FUNCTION_BLOCK FB_PowerNC IMPLEMENTS I_Power
VAR_INPUT
END_VAR
VAR_OUTPUT
END_VAR
VAR
    {attribute 'no_copy'}
    AxisRef : REFERENCE TO AXIS_REF;
    fbMcPower : MC_Power;
    bEnable	: BOOL;
    bEnablePositive : BOOL;
    bEnableNegative : BOOL;
    bPowerIsEnabled : BOOL;
    bBusy 		: BOOL;
    bError 	: BOOL;
    nErrorID 	: UDINT;
    fOverride 	: LREAL := 100.0;
    sMessage : T_MAXSTRING;
    eBufferMode : MC_BufferMode := MC_BufferMode.MC_Aborting;
END_VAR

PROPERTY Aborted : BOOL
GET
END_GET
END_PROPERTY

PROPERTY Active : BOOL
GET
Active := THIS^.bPowerIsEnabled;
END_GET
END_PROPERTY

PROPERTY Busy : BOOL
GET
Busy := THIS^.bBusy;
END_GET
END_PROPERTY

METHOD PUBLIC CallAfterInit
VAR_INPUT
    AxisRef : REFERENCE TO AXIS_REF;
END_VAR
THIS^.AxisRef REF= AxisRef;
END_METHOD

PROPERTY Done : BOOL
GET
END_GET
END_PROPERTY

METHOD Enables
VAR_INPUT
    Enable	: BOOL;
    Enable_Positive	: BOOL;
    Enable_Negative	: BOOL;
END_VAR
THIS^.bEnable := Enable;
THIS^.bEnablePositive := Enable_Positive;
THIS^.bEnableNegative := Enable_Negative;
END_METHOD

PROPERTY Error : BOOL
GET
Error := bError;
END_GET
END_PROPERTY

PROPERTY ErrorID : UDINT
GET
ErrorID := nErrorID;
END_GET
END_PROPERTY

//FB_Init is always available implicitly and it is used primarily for initialization.
//The return value is not evaluated. For a specific influence, you can also declare the
//methods explicitly and provide additional code there with the standard initialization
//code. You can evaluate the return value.
METHOD FB_Init: BOOL
VAR_INPUT
    bInitRetains: BOOL; // TRUE: the retain variables are initialized (reset warm / reset cold)
    bInCopyCode: BOOL;  // TRUE: the instance will be copied to the copy code afterward (online change)
    AxisRef : REFERENCE TO AXIS_REF;
END_VAR
THIS^.AxisRef REF= AxisRef;
END_METHOD

PROPERTY Message : T_MAXSTRING
GET
Message := sMessage;
END_GET
END_PROPERTY

PROPERTY Override : LREAL
GET
Override := THIS^.fOverride;
END_GET
END_PROPERTY

METHOD Power
VAR_INPUT
    Enable	: BOOL;
    Enable_Positive	: BOOL;
    Enable_Negative	: BOOL;
    Override	: LREAL := 100.0;
    BufferMode	: MC_BufferMode := MC_BufferMode.MC_Aborting;
END_VAR
THIS^.bEnable := Enable;
THIS^.bEnablePositive := Enable_Positive;
THIS^.bEnableNegative := Enable_Negative;
THIS^.fOverride := Override;
THIS^.eBufferMode := BufferMode ;
END_METHOD

PROPERTY PowerIsEnabled : BOOL
GET
PowerIsEnabled := bPowerIsEnabled;
END_GET
END_PROPERTY

END_FUNCTION_BLOCK

(* stored: Version 1.1.0.1
   POU FB_PowerNC: Id {82bac45d-f3fb-4090-96f5-9cec57f017c8}, SpecialFunc None
   Property Aborted: Id {bde69de1-325d-451d-b0a6-8cb993ec4d33}
   Get Get: Id {8c49db22-f93b-4013-b841-4a43a6216501}
   Property Active: Id {49693f07-c88b-4b06-be0c-0dc75c8f5fac}
   Get Get: Id {b11a8d39-0dfc-40d5-ab4e-e7fe1f8bda7c}
   Property Busy: Id {1d88cc85-9bbc-4836-b583-4a9d93ccadc7}
   Get Get: Id {e8b60715-a1d9-4e57-9f76-50ea68243628}
   Method CallAfterInit: Id {b807f150-fc9f-4aa5-9d8d-b294c818c5aa}
   Property Done: Id {47775ab2-32ed-415e-8f00-7dc8c50e6589}
   Get Get: Id {8a26bdf6-610d-44e7-af87-ff96e882b31e}
   Method Enables: Id {60dea20e-362a-45d5-ab02-9c322c575503}
   Property Error: Id {5900c701-bb24-4682-9d2c-47b8d2773b46}
   Get Get: Id {50fb1906-033c-485b-9e5d-f1230f94dfc8}
   Property ErrorID: Id {1fe914ad-7f24-41a0-bde2-d4d693aeb73f}
   Get Get: Id {8f8eef06-c2be-4844-866a-ef0542739cd8}
   Method FB_Init: Id {cf7caa46-f1e4-49f9-addf-eba93ec02164}
   Property Message: Id {8449188f-1930-49b3-8fe2-2e40bd14ae5f}
   Get Get: Id {1b9ef192-6b77-407c-a88f-8d85eb8cdc1a}
   Property Override: Id {a7a1e83f-16ea-4038-8048-9acd1171492b}
   Get Get: Id {c098132b-e311-41da-b640-f143b09d83d2}
   Method Power: Id {b859403c-f315-4c59-bb46-554245f47326}
   Property PowerIsEnabled: Id {7e136934-4440-48f5-a211-011704d8f4f5}
   Get Get: Id {fffb35ff-b9f5-44f8-bd6c-842b697893c4} *)
